// TIA Portal V20 export
TYPE "typeEmHomedCheck"
// stored: Access Published, Namespace Unit1.Em5
   STRUCT
      cmNgAndManualInputAxisY : Bool;
      cmMagazineAxisZ : Bool;
      cmNgAndManualInputCylinderUpDown : Bool;
      cmNgAndManualInputVacuumUnit : Bool;
      cmNgAndManualInputVibratorUnit : Bool;
      cmMagazineLockCylinderUpDown : Bool;
   END_STRUCT;
END_TYPE
